IO10: NOP   0;
      NOP   0;
// --- FCM 11 - Floor drives and lifting devices and screw ---
      L     "MAL1S033Par".Ilo.ILOMode;
      L     11;
      <>I   ;
      SPB   IO11;
// man on
      U     "MAL1S033Par".Ilo.GrCMDManOn[1];
      S     "G291M".Gr.InManual; // LIFTING DEVICE KILN 2
      S     "G291M".Gr.CmdOn; // No Button: LIFTING DEVICE KILN 2
      S     "G291M".Gr.CmdContinue; // No Button LIFTING DEVICE KILN 2
      S     "G292M".Gr.InManual; // TRAVELLING DRIVE KILN 2
      S     "G293M".Gr.InManual; // UNLOADING / LOADING SCREW KILN 2
      R     "MAL1S033Par".Ilo.GrCMDManOn[1];
// man off
      U     "MAL1S033Par".Ilo.GrCMDManOff[1];
      S     "G291M".Gr.CmdManualOff; // LIFTING DEVICE KILN 2
      R     "G291M".Gr.InManual; // LIFTING DEVICE KILN 2
      R     "G291M".USW14; // ILO-cmd
      R     "G291M".USW15; // ILO-cmd
      S     "G292M".Gr.CmdManualOff; // TRAVELLING DRIVE KILN 2
      R     "G292M".Gr.InManual; // TRAVELLING DRIVE KILN 2
      R     "G292M".USW14; // ILO-cmd
      R     "G292M".USW15; // ILO-cmd
      S     "G293M".Gr.CmdManualOff; // UNLOADING / LOADING SCREW KILN 2
      R     "G293M".Gr.InManual; // UNLOADING / LOADING SCREW KILN 2
      R     "G293M".USW14; // ILO-cmd
      R     "G293M".USW15; // ILO-cmd
      R     "MAL1S033Par".Ilo.GrCMDManOff[1];
      R     "MAL1S033Par".Ilo.GrCMDManAdditional.Cmd1[1];
      R     "MAL1S033Par".Ilo.GrCMDManAdditional.Cmd2[1];
// man start
      U     "MAL1S033Par".Ilo.GrCMDManStart[1];
      S     "G292M".Gr.CmdOn; // TRAVELLING DRIVE KILN 2
      S     "G292M".Gr.CmdContinue; // TRAVELLING DRIVE KILN 2
      R     "MAL1S033Par".Ilo.GrCMDManStart[1];
      U     "MAL1S033Par".Ilo.GrCMDManStart[2];
      S     "G291M".Gr.CmdOn; // LIFTING DEVICE KILN 2
      S     "G291M".Gr.CmdContinue; // LIFTING DEVICE KILN 2
      R     "MAL1S033Par".Ilo.GrCMDManStart[2];
      U     "MAL1S033Par".Ilo.GrCMDManStart[3];
      S     "G293M".Gr.CmdOn; // UNLOADING / LOADING SCREW KILN 2
      S     "G293M".Gr.CmdContinue; // UNLOADING / LOADING SCREW KILN 2
      R     "MAL1S033Par".Ilo.GrCMDManStart[3];
//MW 2010.04.26      U     "MAL1S033Par".Ilo.GrCMDManStart[4]
//MW 2010.04.26      S     "G293M".Gr.CmdOn            // UNLOADING / LOADING SCREW KILN 2
//MW 2010.04.26      S     "G293M".Gr.CmdContinue      // UNLOADING / LOADING SCREW KILN 2
//MW 2010.04.26      R     "MAL1S033Par".Ilo.GrCMDManStart[4]
// man stop
      U     "MAL1S033Par".Ilo.GrCMDManStop[1];
      S     "G291M".Gr.CmdOff; // LIFTING DEVICE KILN 2
      S     "G292M".Gr.CmdOff; // TRAVELLING DRIVE KILN 2
      S     "G293M".Gr.CmdOff; // UNLOADING / LOADING SCREW KILN 2
      R     "MAL1S033Par".Ilo.GrCMDManStop[1];
// man fault reset
      U     "MAL1S033Par".Ilo.GrCMDManFaultReset[1];
      S     "G291M".Gr.CmdFaultReset; // LIFTING DEVICE KILN 2
      S     "G292M".Gr.CmdFaultReset; // TRAVELLING DRIVE KILN 2
      S     "G293M".Gr.CmdFaultReset; // UNLOADING / LOADING SCREW KILN 2
      R     "MAL1S033Par".Ilo.GrCMDManFaultReset[1];
// moving direction
      UN    "G292M".Gr.InManual; // TRAVELLING DRIVE KILN 2
      O     ;
      UN    "MAL1S033Par".Ilo.GrCMDManAdditional.Cmd1[1];
      UN    "MAL1S033Par".Ilo.GrCMDManAdditional.Cmd2[1];
      SPB   f112;
      U     "MAL1S033Par".Ilo.GrCMDManAdditional.Cmd1[1];
      =     "G292M".USW14; // ILO-cmd run fwd
      U     "MAL1S033Par".Ilo.GrCMDManAdditional.Cmd2[1];
      =     "G292M".USW15; // ILO-cmd run rev
// target speed floor drives
      L     "MAL1S033Par".Ilo.SetpointInt01[1];
      T     "MAL1S033Par".Par.ParIntProcess.Speed_ILO_FloorRotating;
f112: NOP   0;
      UN    "G291M".Gr.InManual; // Malting Plant OAO Belsolod Ivanonvo Weissrussland
      O(    ;
      L     "MAL1S033Par".Ilo.Code_ILO_Funktion0;
      L     1100;
      <>I   ;
      )     ;
      SPB   f113;
// target position lifting devices
      L     "MAL1S033Par".Ilo.SetpointInt01[2];
      L     "MAL1S033Par".Ilo.SetpointInt02[1];
      T     "MAL1S033Par".Par.ParIntProcess.TarPos_ILO_LiftDev;
f113: NOP   0;
      UN    "G293M".Gr.InManual; // UNLOADING / LOADING SCREW KILN 2
      O     ;
      UN    "MAL1S033Par".Ilo.GrCMDManAdditional.Cmd1[3];
      UN    "MAL1S033Par".Ilo.GrCMDManAdditional.Cmd2[3];
      SPB   f114;
      U     "MAL1S033Par".Ilo.GrCMDManAdditional.Cmd1[3];
      =     "G293M".USW14; // ILO-cmd run fwd
      U     "MAL1S033Par".Ilo.GrCMDManAdditional.Cmd2[3];
      =     "G293M".USW15; // ILO-cmd run rev
f114: NOP   0;
IO11: NOP   0;
      NOP   0;
// --- FCM 12 - Floor drives and lifting devices and screw and discharging flap ---
      L     "MAL1S033Par".Ilo.ILOMode;
      L     12;
      <>I   ;
      SPB   IO12;
// man on
      U     "MAL1S033Par".Ilo.GrCMDManOn[1];
      S     "G291M".Gr.InManual; // LIFTING DEVICE KILN 2
      S     "G291M".Gr.CmdOn; // No Button: LIFTING DEVICE KILN 2
      S     "G291M".Gr.CmdContinue; // No Button LIFTING DEVICE KILN 2
      S     "G292M".Gr.InManual; // TRAVELLING DRIVE KILN 2
      S     "G293M".Gr.InManual; // UNLOADING / LOADING SCREW KILN 2
      S     "G294M".Gr.InManual; // DISCHARGE DOOR KILN 2
      R     "MAL1S033Par".Ilo.GrCMDManOn[1];
// man off
      U     "MAL1S033Par".Ilo.GrCMDManOff[1];
      S     "G291M".Gr.CmdManualOff; // LIFTING DEVICE KILN 2
      R     "G291M".Gr.InManual; // LIFTING DEVICE KILN 2
      R     "G291M".USW14; // ILO-cmd
      R     "G291M".USW15; // ILO-cmd
      S     "G292M".Gr.CmdManualOff; // TRAVELLING DRIVE KILN 2
      R     "G292M".Gr.InManual; // TRAVELLING DRIVE KILN 2
      R     "G292M".USW14; // ILO-cmd
      R     "G292M".USW15; // ILO-cmd
      S     "G293M".Gr.CmdManualOff; // UNLOADING / LOADING SCREW KILN 2
      R     "G293M".Gr.InManual; // UNLOADING / LOADING SCREW KILN 2
      R     "G293M".USW14; // ILO-cmd
      R     "G293M".USW15; // ILO-cmd
      S     "G294M".Gr.CmdManualOff; // DISCHARGE DOOR KILN 2
      R     "G294M".Gr.InManual; // DISCHARGE DOOR KILN 2
      R     "G294M".USW14; // ILO-cmd
      R     "G294M".USW15; // ILO-cmd
      R     "MAL1S033Par".Ilo.GrCMDManOff[1];
      R     "MAL1S033Par".Ilo.GrCMDManAdditional.Cmd1[1];
      R     "MAL1S033Par".Ilo.GrCMDManAdditional.Cmd2[1];
// man start
      U     "MAL1S033Par".Ilo.GrCMDManStart[1];
      S     "G292M".Gr.CmdOn; // TRAVELLING DRIVE KILN 2
      S     "G292M".Gr.CmdContinue; // TRAVELLING DRIVE KILN 2
      R     "MAL1S033Par".Ilo.GrCMDManStart[1];
      U     "MAL1S033Par".Ilo.GrCMDManStart[2];
      S     "G291M".Gr.CmdOn; // LIFTING DEVICE KILN 2
      S     "G291M".Gr.CmdContinue; // LIFTING DEVICE KILN 2
      R     "MAL1S033Par".Ilo.GrCMDManStart[2];
      U     "MAL1S033Par".Ilo.GrCMDManStart[3];
      S     "G293M".Gr.CmdOn; // UNLOADING / LOADING SCREW KILN 2
      S     "G293M".Gr.CmdContinue; // UNLOADING / LOADING SCREW KILN 2
      R     "MAL1S033Par".Ilo.GrCMDManStart[3];
      U     "MAL1S033Par".Ilo.GrCMDManStart[4];
//MW 2010.04.26      S     "G293M".Gr.CmdOn            // UNLOADING / LOADING SCREW KILN 2
//MW 2010.04.26      S     "G293M".Gr.CmdContinue      // UNLOADING / LOADING SCREW KILN 2
      S     "G294M".Gr.CmdOn; // DISCHARGE DOOR KILN 2
      S     "G294M".Gr.CmdContinue; // DISCHARGE DOOR KILN 2
      R     "MAL1S033Par".Ilo.GrCMDManStart[4];
// man stop
      U     "MAL1S033Par".Ilo.GrCMDManStop[1];
      S     "G291M".Gr.CmdOff; // LIFTING DEVICE KILN 2
      S     "G292M".Gr.CmdOff; // TRAVELLING DRIVE KILN 2
      S     "G293M".Gr.CmdOff; // UNLOADING / LOADING SCREW KILN 2
      S     "G294M".Gr.CmdOff; // DISCHARGE DOOR KILN 2
      R     "MAL1S033Par".Ilo.GrCMDManStop[1];
// man fault reset
      U     "MAL1S033Par".Ilo.GrCMDManFaultReset[1];
      S     "G291M".Gr.CmdFaultReset; // LIFTING DEVICE KILN 2
      S     "G292M".Gr.CmdFaultReset; // TRAVELLING DRIVE KILN 2
      S     "G293M".Gr.CmdFaultReset; // UNLOADING / LOADING SCREW KILN 2
      S     "G294M".Gr.CmdFaultReset; // DISCHARGE DOOR KILN 2
      R     "MAL1S033Par".Ilo.GrCMDManFaultReset[1];
// moving direction
      UN    "G292M".Gr.InManual; // TRAVELLING DRIVE KILN 2
      O     ;
      UN    "MAL1S033Par".Ilo.GrCMDManAdditional.Cmd1[1];
      UN    "MAL1S033Par".Ilo.GrCMDManAdditional.Cmd2[1];
      SPB   f122;
      U     "MAL1S033Par".Ilo.GrCMDManAdditional.Cmd1[1];
      =     "G292M".USW14; // ILO-cmd run fwd
      U     "MAL1S033Par".Ilo.GrCMDManAdditional.Cmd2[1];
      =     "G292M".USW15; // ILO-cmd run rev
// target speed floor drives
      L     "MAL1S033Par".Ilo.SetpointInt01[1];
      T     "MAL1S033Par".Par.ParIntProcess.Speed_ILO_FloorRotating;
f122: NOP   0;
      UN    "G291M".Gr.InManual; // LIFTING DEVICE KILN 2
      O(    ;
      L     "MAL1S033Par".Ilo.Code_ILO_Funktion0;
      L     1200;
      <>I   ;
      )     ;
      SPB   f123;
// target position lifting devices
      L     "MAL1S033Par".Ilo.SetpointInt02[1];
      T     "MAL1S033Par".Par.ParIntProcess.TarPos_ILO_LiftDev;
f123: NOP   0;
      UN    "G293M".Gr.InManual; // Malting Plant OAO Belsolod Ivanonvo Weissrussland
      O     ;
      UN    "MAL1S033Par".Ilo.GrCMDManAdditional.Cmd1[3];
      UN    "MAL1S033Par".Ilo.GrCMDManAdditional.Cmd2[3];
      SPB   f124;
      U     "MAL1S033Par".Ilo.GrCMDManAdditional.Cmd1[3];
//JV070810      =     "G293M".USW14               // ILO-cmd run fwd
      =     "G293M".USW15; // ILO-cmd run rev  //JV070810 nur entladen
      R     "G293M".USW14; // ILO-cmd run fwd  //JV070810 nur entladen
      U     "MAL1S033Par".Ilo.GrCMDManAdditional.Cmd2[3];
      =     "G293M".USW15; // ILO-cmd run rev  //JV070810 nur entladen
      R     "G293M".USW14; // ILO-cmd run fwd  //JV070810 nur entladen

f124: NOP   0;
      UN    "G294M".Gr.InManual; // DISCHARGE DOOR KILN 2
      O     ;
      UN    "MAL1S033Par".Ilo.GrCMDManAdditional.Cmd1[4];
      UN    "MAL1S033Par".Ilo.GrCMDManAdditional.Cmd2[4];
      SPB   f125;
      U     "MAL1S033Par".Ilo.GrCMDManAdditional.Cmd1[4];
      =     "G294M".USW14; // ILO-cmd OPEN
      U     "MAL1S033Par".Ilo.GrCMDManAdditional.Cmd2[4];
      =     "G294M".USW15; // ILO-cmd CLOSE
f125: NOP   0;
IO12: NOP   0;
//
// copy state
      U     "G291M".Gr.InOutAutostartMan; // LIFTING DEVICE KILN 2
      =     "MAL1S033Par".Ilo.GrSTMan[1];
      U     "G292M".Gr.InOutAutostartMan; // TRAVELLING DRIVE KILN 2
      =     "MAL1S033Par".Ilo.GrSTMan[2];
      U     "G293M".Gr.InOutAutostartMan; // UNLOADING / LOADING SCREW KILN 2
      =     "MAL1S033Par".Ilo.GrSTMan[3];
      U     "G294M".Gr.InOutAutostartMan; // DISCHARGE DOOR KILN 2
      =     "MAL1S033Par".Ilo.GrSTMan[4];
      U     "G297M".Gr.InOutAutostartMan; // FAN KILN 2
      =     "MAL1S033Par".Ilo.GrSTMan[6];
      U     "G302M".Gr.InOutAutostartMan; // HEATING KILN 2
      =     "MAL1S033Par".Ilo.GrSTMan[11];
      U     "G303M".Gr.InOutAutostartMan; // LOUVER AIR HEATER KILN 2
      =     "MAL1S033Par".Ilo.GrSTMan[12];
      U     "G298M".Gr.InOutAutostartMan; // FRESH AIR LOUVER KILN 2
      =     "MAL1S033Par".Ilo.GrSTMan[13];
      U     "G304M".Gr.InOutAutostartMan; // WITHERING AIR KILN 2
      =     "MAL1S033Par".Ilo.GrSTMan[14];
      U     "G299M".Gr.InOutAutostartMan; // RECYCLING AIR FLAP KILN 2
      =     "MAL1S033Par".Ilo.GrSTMan[15];
      U     "G279M".Gr.InOutAutostartMan; // HEATING KILN 1 + 2
      =     "MAL1S033Par".Ilo.GrSTMan[16];
NETWORK
TITLE =ASW_9999: Init Flag
// clear all flags explicde to find them back
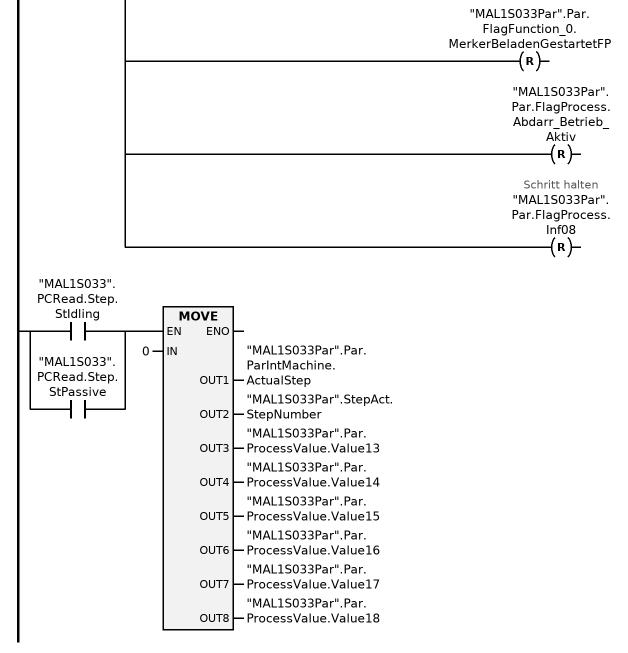
      U     "MAL1S033".PCRead.Step.StIdling;
      O     "MAL1S033".PCRead.Step.StPassive;
      R     "MAL1S033Par".Par.FlagFunction_1.StepLoading;
      R     "MAL1S033Par".Par.FlagFunction_1.StepUnloading;
      R     "MAL1S033Par".Par.FlagFunction_1.StepCleaning;
      R     "MAL1S033Par".Par.FlagFunction_1.LoadingBreak;
      R     "MAL1S033Par".Par.FlagFunction_1.UnloadingBreak;
      R     "MAL1S033Par".Par.FlagFunction_1.CleaningBreak;
      R     "MAL1S033Par".Par.FlagFunction_1.FinishLoading;
      R     "MAL1S033Par".Par.FlagFunction_1.FinishUnloading;
      R     "MAL1S033Par".Par.FlagFunction_1.FinishCleaning;
      R     "MAL1S033Par".Par.FlagFunction_1.Entladerunden_erreicht;
      R     "MAL1S033Par".Par.FlagFunction_1.Reinigungsrunde_erreicht;
      R     "MAL1S033Par".Par.FlagFunction_1.UnloadEnd;
      R     "MAL1S033Par".Par.FlagFunction_1.LoadEnd;
      R     "MAL1S033Par".Par.FlagFunction_1.UnloadFirstPart;
      R     "MAL1S033Par".Par.FlagFunction_1.UnloadSecondPart;
      R     "MAL1S033Par".Par.FlagProcess.ProcessActive;
      R     "MAL1S033Par".Par.FlagProcess.StartProzess_FP;
      R     "MAL1S033Par".Par.FlagProcess.StartProzess_SCAN;
      R     "MAL1S033Par".Par.FlagProcess.TurningFloor;
      R     "MAL1S033Par".Par.FlagProcess.Cooling_Activ;
      R     "MAL1S033Par".Par.FlagProcess.FP_SendResultToPIC;
      R     "MAL1S033Par".Par.FlagProcess.ProcessEnd;

// --> Wie bei Bank Avangard
//MW 2010.04.06
      U     "MAL1S033".PCRead.Step.StPassive;
      R     "MAL1S033Par".Par.FlagMachine.WEGMESSUNG_0_FLAG;
      R     "MAL1S033Par".Par.FlagMachine.ImpulsNullstellung;
      R     "MAL1S033Par".Par.FlagMachine.CmdTurnFwdAfterLoading;
      R     "MAL1S033Par".Par.FlagMachine.CmdTurnRevAfterLoading;
      R     "MAL1S033Par".Par.FlagMachine.ImpulsNullstellungFP;
      R     "MAL1S033Par".Par.FlagMachine.CmdTurnFwdAfterTurning;
      R     "MAL1S033Par".Par.FlagMachine.CmdTurnRevAfterTurning;
      R     "MAL1S033Par".Par.FlagMachine.WEGMESSUNG_0;
      R     "MAL1S033Par".Par.FlagMachine.CmdTurnFwdAfterUnloading;
      R     "MAL1S033Par".Par.FlagMachine.CmdTurnRevAfterUnloading;
      R     "MAL1S033Par".Par.FlagMachine.NULL_INDEX_FP;
      R     "MAL1S033Par".Par.FlagFunction_0.MerkerBeladenGestartetFP;
      R     "MAL1S033Par".Par.FlagProcess.Abdarr_Betrieb_Aktiv;
      R     "MAL1S033Par".Par.FlagProcess.Inf08; // Schritt halten
//
      U     "MAL1S033".PCRead.Step.StIdling;
      O     "MAL1S033".PCRead.Step.StPassive;
      SPBN  csn;
      L     0; // clear step number
      T     "MAL1S033Par".Par.ParIntMachine.ActualStep;
      T     "MAL1S033Par".StepAct.StepNumber;
      T     "MAL1S033Par".Par.ProcessValue.Value13; // Schaltpunkt Regelung
      T     "MAL1S033Par".Par.ProcessValue.Value14; // Sollwert Umluftklappen Kühlen
      T     "MAL1S033Par".Par.ProcessValue.Value15; // Sollwert Ventilator Kühlen
      T     "MAL1S033Par".Par.ProcessValue.Value16; // Step-Copy
      T     "MAL1S033Par".Par.ProcessValue.Value17; // Sollwert Umluftklappen Verbund
      T     "MAL1S033Par".Par.ProcessValue.Value18; // Sollwert Ventilator Verbund

csn:  NOP   0;

NETWORK
TITLE =Main0_End: Init flag
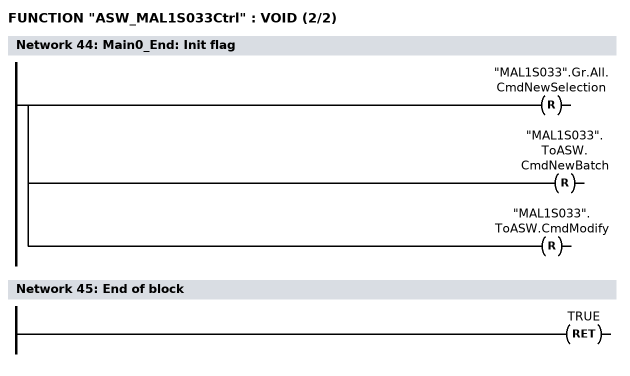

      SET   ;
      R     "MAL1S033".Gr.All.CmdNewSelection;
      R     "MAL1S033".ToASW.CmdNewBatch;
      R     "MAL1S033".ToASW.CmdModify;

NETWORK
TITLE =End of block

      BE    ;

END_FUNCTION

